FUNCTION_BLOCK FB_ComplementaryFilter
VAR_INPUT
    stAccelData : ST_3D_values; // Acceleration Data in (g)
    stGyroData : ST_3D_values; // Gyroscope Data in (°/s)
    fCycleTime : REAL; // Cycle Time (s)
    fAlpha : REAL := 0.98; // Filter coefficient
    bSetReference : BOOL; // Flag to set reference position
END_VAR

VAR_OUTPUT
    stEulerAngle_deg : ST_3D_values; // Euler angle in degrees X= Pitch, Y=Roll, Z=Yaw
    stEulerAngle_rad : ST_3D_values; // Euler angle in rad X= Pitch, Y=Roll, Z=Yaw
END_VAR

VAR
	stRef_Angles_deg :ST_3d_values; // Reference orientation (bSetReference; angles in degrees)

    fAccAngleRoll : REAL;
    fAccAnglePitch : REAL;
	
    fGyroAngleRoll : REAL;
    fGyroAnglePitch : REAL;
    fGyroAngleYaw : REAL;
END_VAR

// Calculate accelerometer angles using ATAN2, which returns radians
IF ((stAccelData.X * stAccelData.X + stAccelData.Z * stAccelData.Z)> 0.0) THEN 	
	fAccAngleRoll := ATAN2(stAccelData.Y, SQRT(stAccelData.X * stAccelData.X + stAccelData.Z * stAccelData.Z));
END_IF
IF ((stAccelData.Y * stAccelData.Y + stAccelData.Z * stAccelData.Z)> 0.0) THEN
	fAccAnglePitch := ATAN2(-stAccelData.X, SQRT(stAccelData.Y * stAccelData.Y + stAccelData.Z * stAccelData.Z));
END_IF

// Convert gyroscope rates from °/s to rad/s before integration
stGyroData.X := stGyroData.X * pi / 180.0;
stGyroData.Y := stGyroData.Y * pi / 180.0;
stGyroData.Z := stGyroData.Z * pi / 180.0;

// Integrate gyroscope rates to get angles in radians
fGyroAnglePitch := fGyroAnglePitch + stGyroData.X * fCycleTime;
fGyroAngleRoll := fGyroAngleRoll + stGyroData.Y * fCycleTime;
fGyroAngleYaw := fGyroAngleYaw + stGyroData.Z * fCycleTime;

// Apply complementary filter
stEulerAngle_rad.X := fAlpha * (fGyroAnglePitch) + (1.0 - fAlpha) * fAccAnglePitch;
stEulerAngle_rad.Y := fAlpha * (fGyroAngleRoll) + (1.0 - fAlpha) * fAccAngleRoll;
stEulerAngle_rad.Z := fGyroAngleYaw; // Yaw is integrated directly from gyroscope

// Convert radians to degrees for output
stEulerAngle_deg.X := stEulerAngle_rad.X * 180.0 / pi;
stEulerAngle_deg.Y := stEulerAngle_rad.Y * 180.0 / pi;
stEulerAngle_deg.Z := stEulerAngle_rad.Z * 180.0 / pi;

// Set reference position if flag is active
IF bSetReference THEN
    stRef_Angles_deg.X := stEulerAngle_deg.X;
    stRef_Angles_deg.Y := stEulerAngle_deg.Y;
    stRef_Angles_deg.Z := stEulerAngle_deg.Z;
END_IF

// Apply reference position
stEulerAngle_deg.X := stEulerAngle_deg.X - (stRef_Angles_deg.X);
stEulerAngle_deg.Y := stEulerAngle_deg.Y - (stRef_Angles_deg.Y);
stEulerAngle_deg.Z := stEulerAngle_deg.Z- (stRef_Angles_deg.Z);

stEulerAngle_rad.X := stEulerAngle_rad.X - (stRef_Angles_deg.X) * pi / 180.0;
stEulerAngle_rad.Y := stEulerAngle_rad.Y - (stRef_Angles_deg.Y) * pi / 180.0;
stEulerAngle_rad.Z := stEulerAngle_rad.Z - (stRef_Angles_deg.Z) * pi / 180.0;

END_FUNCTION_BLOCK

(* stored: Version 1.1.0.1, ProductVersion 3.1.4024.13
   POU FB_ComplementaryFilter: Id {b52c30cc-d6ec-4f96-8950-1da13efb107a}, SpecialFunc None *)
